FUNCTION_BLOCK RollerConveyor EXTENDS Conveyor
VAR_INPUT
END_VAR
VAR_OUTPUT
END_VAR
VAR
END_VAR

Super^();

END_FUNCTION_BLOCK

(* stored: Version 1.1.0.1, ProductVersion 3.1.4024.2
   POU RollerConveyor: Id {fea9d20d-0e09-459b-a5ba-bec52b89bada}, SpecialFunc None *)
